SUBAPPLICATION SwitchPic_2_2 (* Bild umschalten VT und AUX; 2 Zustände *)
  (* Standard: 61499-2 *)
  (* Version 1.0, 2026-05-29, franz *)
  PACKAGE MyLib::sys;
  IMPORT isobus::UT::Q::const::IDs::ID_NULL;
  IMPORT isobus::UT::Q::types::s2x1ObjectIDs;
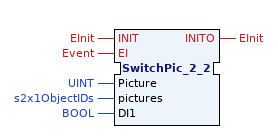
  EVENT_INPUT
    INIT : EInit; (* Initialization Request *)
    EI;
  END_EVENT
  EVENT_OUTPUT
    INITO : EInit; (* Initialization Confirm *)
  END_EVENT
  VAR_INPUT
    Picture : UINT := ID_NULL; (* Object ID of the ObjectPointer to the Picture *)
    pictures : isobus::UT::Q::types::s2x1ObjectIDs := (up := (u16ObjId := ID_NULL), down := (u16ObjId := ID_NULL)); (* the single Pictures *)
    DI1 : BOOL := FALSE; (* Selector *)
  END_VAR
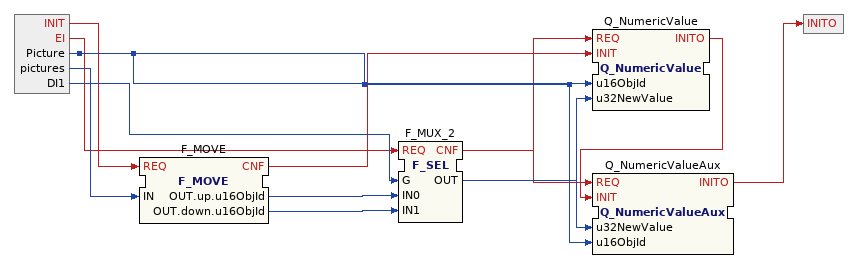
  FBS
    Q_NumericValue : isobus::UT::Q::Q_NumericValue;
    F_MOVE : iec61131::selection::F_MOVE; {SET_ATTRIBUTE(DataType, isobus::UT::Q::types::s2x1ObjectIDs)}
    F_MUX_2 : iec61131::selection::F_SEL;
    Q_NumericValueAux : isobus::UT::Q::Q_NumericValueAux;
  END_FBS
  EVENT_CONNECTIONS
    EI TO F_MUX_2.REQ;
    F_MUX_2.CNF TO Q_NumericValue.REQ;
    INIT TO F_MOVE.REQ;
    F_MOVE.CNF TO Q_NumericValue.INIT;
    F_MUX_2.CNF TO Q_NumericValueAux.REQ;
    Q_NumericValueAux.INITO TO INITO;
    Q_NumericValue.INITO TO Q_NumericValueAux.INIT;
  END_CONNECTIONS
  DATA_CONNECTIONS
    Picture TO Q_NumericValue.u16ObjId;
    pictures TO F_MOVE.IN;
    DI1 TO F_MUX_2.G;
    F_MUX_2.OUT TO Q_NumericValue.u32NewValue;
    F_MOVE.OUT.up.u16ObjId TO F_MUX_2.IN0;
    F_MOVE.OUT.down.u16ObjId TO F_MUX_2.IN1;
    F_MUX_2.OUT TO Q_NumericValueAux.u32NewValue;
    Picture TO Q_NumericValueAux.u16ObjId;
  END_CONNECTIONS
END_SUBAPPLICATION
